(* Logix 5000 project; controller Modbus_TCP_Client_Example vendor 1 type 14 code 154 rev 32.15; software revision 32.05; part 5 of 10 *)

ADD_ON_INSTRUCTION AMP_Normal_Stop   (* revision 1.0 *)
// Applied Motion - Stop/Kill using Normal Deceleration - AOI
// Help:
// The Normal Stop AOI is used to stop and kill the drive using the normal deceleration set by the DE command.
VAR_IN_OUT
   Input : DINT[14]; {required}   // Drive Input Assembly
   Output : DINT[16]; {required}   // Drive Output Assembly
        [0]   // Command Word
        [10]   // Data/Register 1
        [11]   // Data/Register 2
        [1]   // Jog Speed (0.25 rev/min)
        [2]   // Jog Acceleration (10 rev/s/s)
        [3]   // Jog Deceleration (10 rev/s/s)
        [4]   // Point-to-Point Velocity (0.25 rev/min)
        [5]   // Point-to-Point Acceleration (10 rev/s/s)
        [6]   // Point-to-Point Deceleration (10 rev/s/s)
        [7]   // Point-to-Point Distance (Motor steps)
        [9]   // (2x ASCII Letters in 16 lower word)
END_VAR
VAR_INPUT
   RPI : DINT := 100; {visible}   // Drive Connection Request Packet Interval (milliseconds)
   Stop : BOOL; {required}   // Stop the drive axis
END_VAR
VAR_OUTPUT
   Sent : BOOL; {access Read Only, visible}   // Stop has been sent to drive
   In_Progress : BOOL; {access Read Only, visible}   // Stop in progress
   Done : BOOL; {access Read Only, visible}   // Stop completed without errors - Servo is not moving
   Error : BOOL; {access Read Only, visible}   // Stop failed - drive not ready or faulted
   State : DINT := 10; {access None}   // Internal state of progress
END_VAR
VAR
   Loc_StatusCode : AMP_Status_Word;
   Loc_CommandOff_Timer : TIMER;   // Timer to make sure command value was 0 before sending a new command
   Loc_CommandOn_Timer : TIMER;   // Timer to make sure command value is set long enough to be sent to servo
   Loc_Input_Assembly : AMP_Input_Assembly_v2; {access None}
   Loc_Stop_ONS : BOOL; {access None}
END_VAR

ROUTINE Logic   (* ladder *)
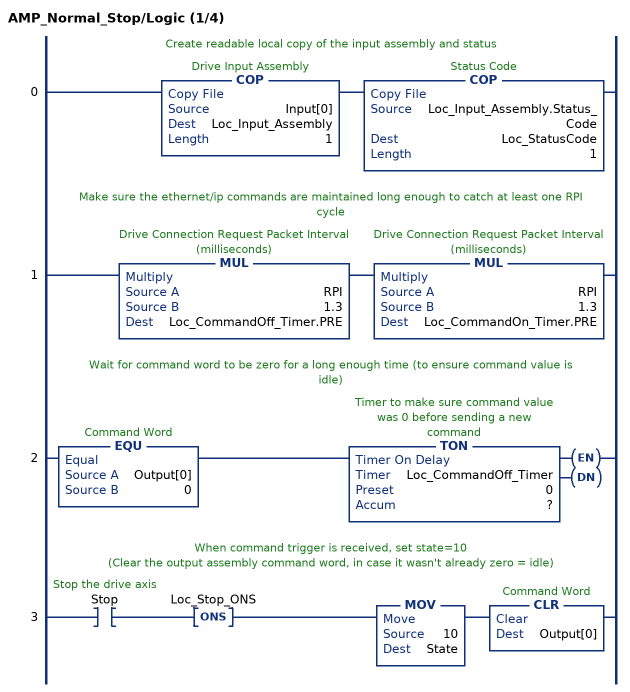
   // Create readable local copy of the input assembly and status
   0: COP(Input[0],Loc_Input_Assembly,1)COP(Loc_Input_Assembly.Status_Code,Loc_StatusCode,1);
   // Make sure the ethernet/ip commands are maintained long enough to catch at least one RPI cycle
   1: MUL(RPI,1.3,Loc_CommandOff_Timer.PRE)MUL(RPI,1.3,Loc_CommandOn_Timer.PRE);
   // Wait for command word to be zero for a long enough time (to ensure command value is idle)
   2: EQU(Output[0],0)TON(Loc_CommandOff_Timer,?,?);
   // When command trigger is received, set state=10
   // (Clear the output assembly command word, in case it wasn't already zero = idle)
   3: XIC(Stop)ONS(Loc_Stop_ONS)MOV(10,State)CLR(Output[0]);
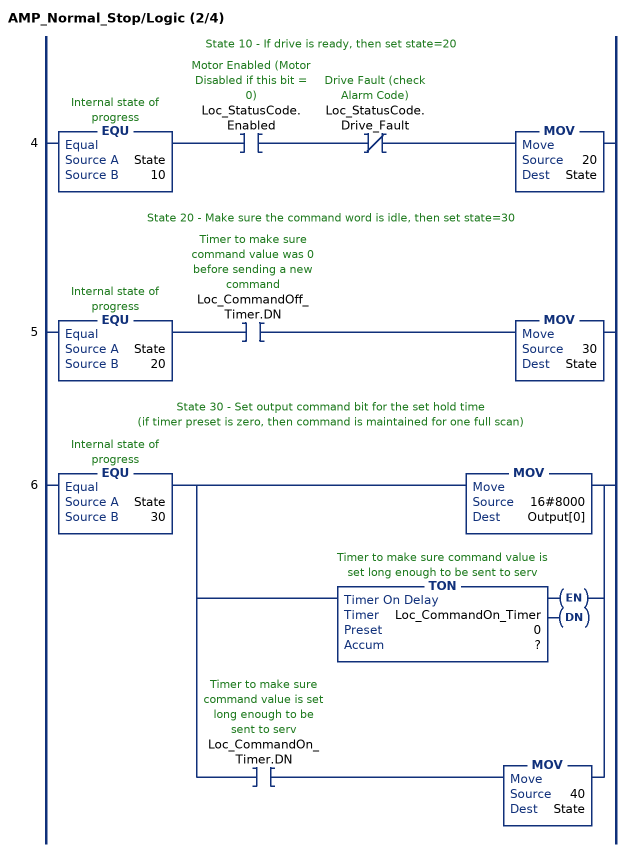
   // State 10 - If drive is ready, then set state=20
   4: EQU(State,10)XIC(Loc_StatusCode.Enabled)XIO(Loc_StatusCode.Drive_Fault)MOV(20,State);
   // State 20 - Make sure the command word is idle, then set state=30
   5: EQU(State,20)XIC(Loc_CommandOff_Timer.DN)MOV(30,State);
   // State 30 - Set output command bit for the set hold time
   // (if timer preset is zero, then command is maintained for one full scan)
   6: EQU(State,30)[MOV(16#8000,Output[0]) ,TON(Loc_CommandOn_Timer,?,?) ,XIC(Loc_CommandOn_Timer.DN) MOV(40,State) ];
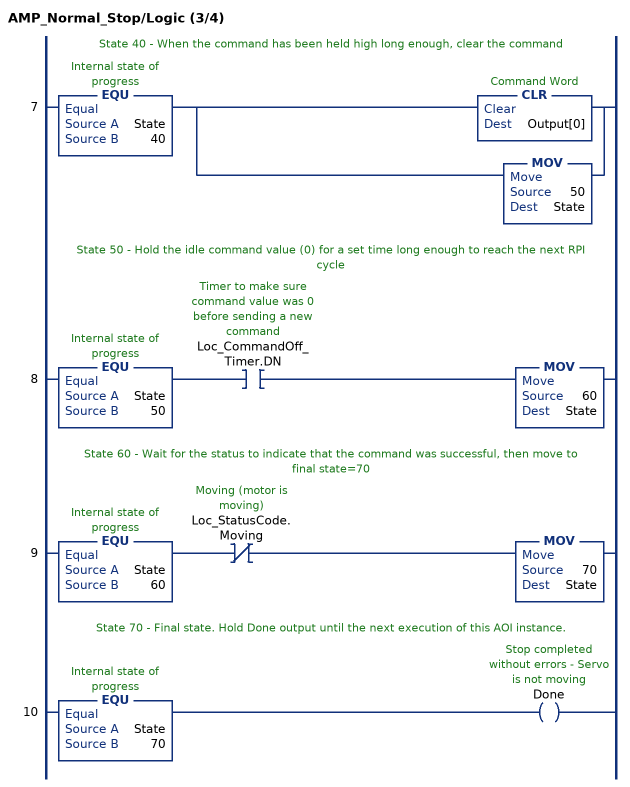
   // State 40 - When the command has been held high long enough, clear the command
   7: EQU(State,40)[CLR(Output[0]) ,MOV(50,State) ];
   // State 50 - Hold the idle command value (0) for a set time long enough to reach the next RPI cycle
   8: EQU(State,50)XIC(Loc_CommandOff_Timer.DN)MOV(60,State);
   // State 60 - Wait for the status to indicate that the command was successful, then move to final state=70
   9: EQU(State,60)XIO(Loc_StatusCode.Moving)MOV(70,State);
   // State 70 - Final state. Hold Done output until the next execution of this AOI instance.
   10: EQU(State,70)OTE(Done);
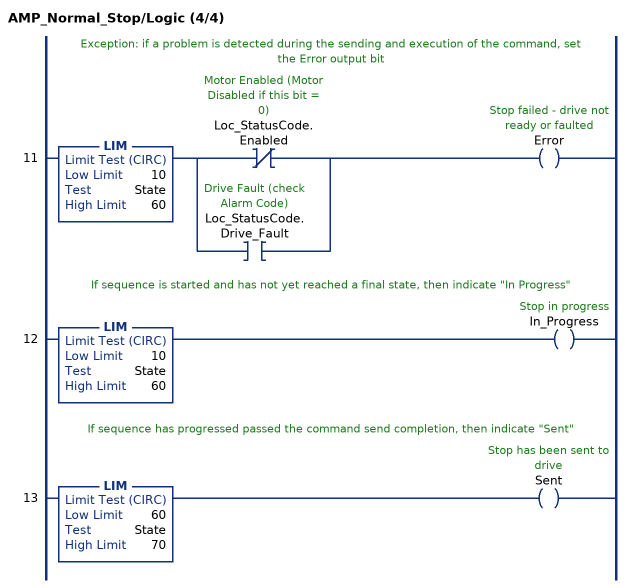
   // Exception: if a problem is detected during the sending and execution of the command, set the Error output bit
   11: LIM(10,State,60)[XIO(Loc_StatusCode.Enabled) ,XIC(Loc_StatusCode.Drive_Fault) ]OTE(Error);
   // If sequence is started and has not yet reached a final state, then indicate "In Progress"
   12: LIM(10,State,60)OTE(In_Progress);
   // If sequence has progressed passed the command send completion, then indicate "Sent"
   13: LIM(60,State,70)OTE(Sent);
END_ROUTINE
END_ADD_ON_INSTRUCTION

ADD_ON_INSTRUCTION AMP_Normal_Stop_Servo   (* revision 1.0, vendor Applied Motion Products Inc. *)
// Applied Motion - Stop/Kill using Normal Deceleration - AOI
// Help:
// This AOI Stops the Motor Jogging/Moving using Deceleration(SKD).
VAR_IN_OUT
   Input : DINT[20]; {required}   // Drive Input Assembly
        [16]   // Analog_Input1
        [4]   // Alarm_Code
        [0]   // Control_Word_Received
        [10]   // Position_Error
        [11]   // Actual_Velocity_RPS
        [12]   // Digital_Outputs
        [13]   // Digital_Inputs
        [14]   // Analog_Output1
        [15]   // Analog_Output2
        [17]   // Analog_Input2
        [18]   // Torque_Limit
        [19]   // Second_Encoder_Speed
        [1]   // OpCode1_Received
        [2]   // Control_Mode
        [3]   // Status_Code
        [5]   // Supply_Voltage
        [6]   // Applied_Torque
        [7]   // Drive_Temperature
        [8]   // Encoder_Position
        [9]   // Second_Encoder_Position
   Output : DINT[11]; {required}   // Drive Output Assembly
        [10]   // Reserved
        [4]   // Target Velocity
        [0]   // Control Word
        [3]   // Target Pos
        [1]   // OpCode 1
        [2]   // OpCode 2
        [5]   // Porifle Acceleration
        [6]   // Profile Deceleration
        [7]   // Target Torque
        [8]   // OpCode 3
        [9]   // OpCode 4
END_VAR
VAR_INPUT
   Stop : BOOL; {required}   // Stop the drive axis (on rising edge)
END_VAR
VAR_OUTPUT
   Sent : BOOL; {access Read Only, visible}   // Stop has been sent to drive
   In_Progress : BOOL; {access Read Only, visible}   // Stop in progress
   Done : BOOL; {access Read Only, visible}   // Stop completed without errors - Servo is not moving
   Error : BOOL; {access Read Only, visible}   // Stop failed - drive not ready or faulted
   State : DINT := 10; {access Read Only}   // Internal state of progress
END_VAR
VAR
   Loc_Stop_ONS : BOOL;
   Loc_StatusCode : AMP_Status_Word_Servo; {access None}
   Loc_Input_Assembly : AMP_Input_Assembly_Servo_v2; {access None}
END_VAR

ROUTINE Logic   (* ladder *)
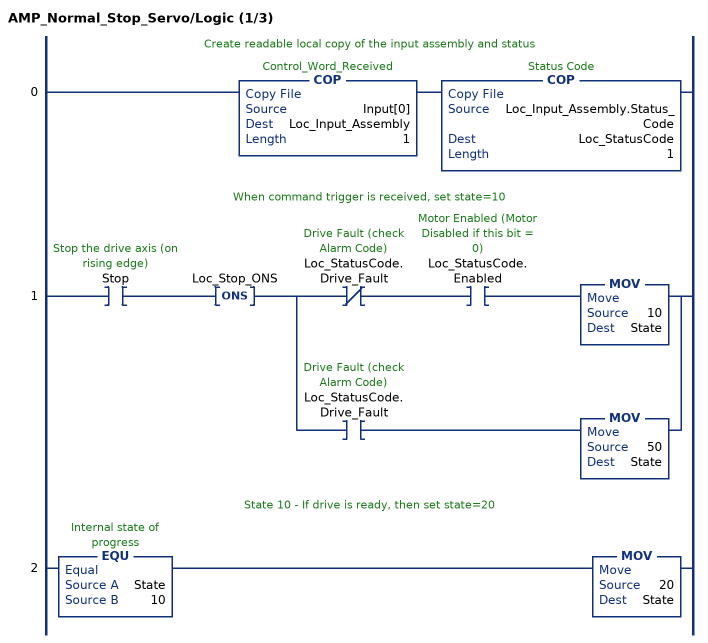
   // Create readable local copy of the input assembly and status
   0: COP(Input[0],Loc_Input_Assembly,1)COP(Loc_Input_Assembly.Status_Code,Loc_StatusCode,1);
   // When command trigger is received, set state=10
   1: XIC(Stop)ONS(Loc_Stop_ONS)[XIO(Loc_StatusCode.Drive_Fault) XIC(Loc_StatusCode.Enabled) MOV(10,State) ,XIC(Loc_StatusCode.Drive_Fault) MOV(50,State) ];
   // State 10 - If drive is ready, then set state=20
   2: EQU(State,10)MOV(20,State);
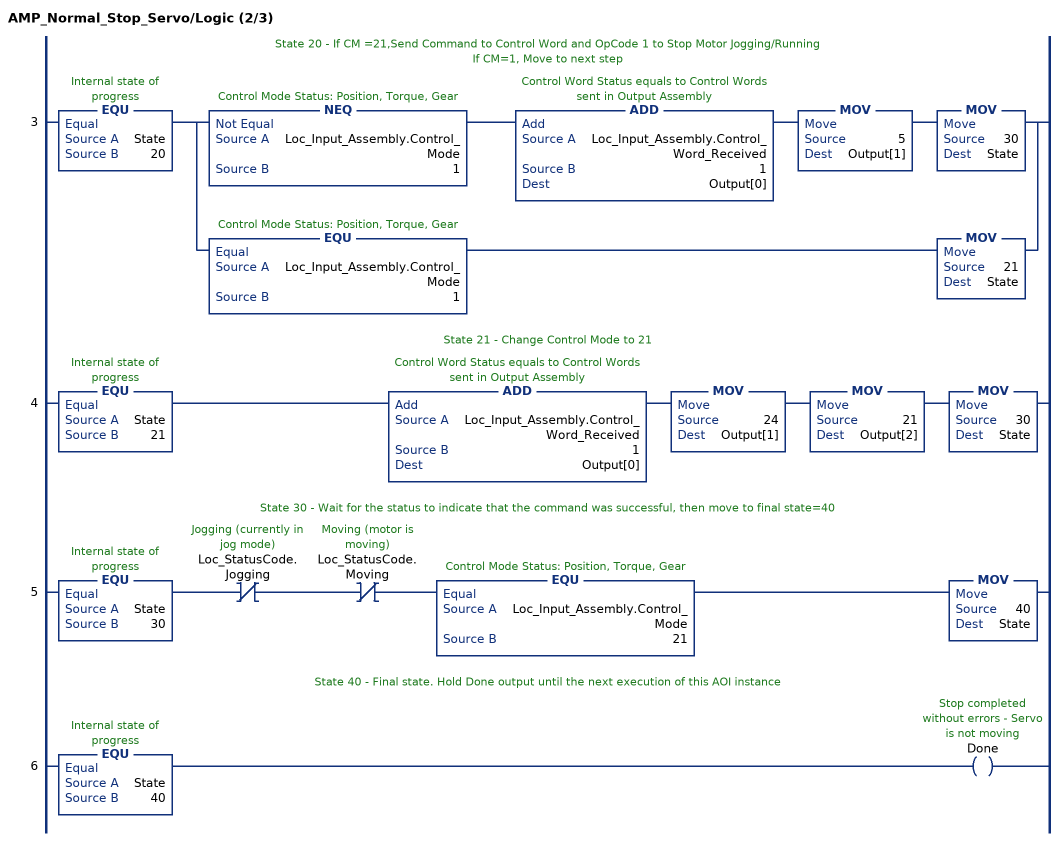
   // State 20 - If CM =21,Send Command to Control Word and OpCode 1 to Stop Motor Jogging/Running
   // If CM=1, Move to next step
   3: EQU(State,20)[NEQ(Loc_Input_Assembly.Control_Mode,1) ADD(Loc_Input_Assembly.Control_Word_Received,1,Output[0]) MOV(5,Output[1]) MOV(30,State) ,EQU(Loc_Input_Assembly.Control_Mode,1) MOV(21,State) ];
   // State 21 - Change Control Mode to 21
   4: EQU(State,21)ADD(Loc_Input_Assembly.Control_Word_Received,1,Output[0])MOV(24,Output[1])MOV(21,Output[2])MOV(30,State);
   // State 30 - Wait for the status to indicate that the command was successful, then move to final state=40
   5: EQU(State,30)XIO(Loc_StatusCode.Jogging)XIO(Loc_StatusCode.Moving)EQU(Loc_Input_Assembly.Control_Mode,21)MOV(40,State);
   // State 40 - Final state. Hold Done output until the next execution of this AOI instance
   6: EQU(State,40)OTE(Done);
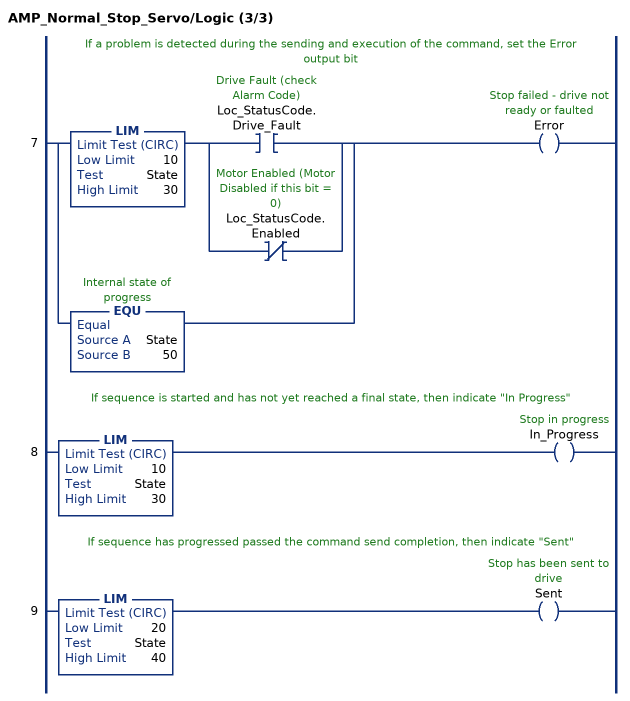
   // If a problem is detected during the sending and execution of the command, set the Error output bit
   7: [LIM(10,State,30) [XIC(Loc_StatusCode.Drive_Fault) ,XIO(Loc_StatusCode.Enabled) ] ,EQU(State,50) ]OTE(Error);
   // If sequence is started and has not yet reached a final state, then indicate "In Progress"
   8: LIM(10,State,30)OTE(In_Progress);
   // If sequence has progressed passed the command send completion, then indicate "Sent"
   9: LIM(20,State,40)OTE(Sent);
END_ROUTINE
END_ADD_ON_INSTRUCTION

ADD_ON_INSTRUCTION AMP_Point_to_Point_FC_Servo   (* revision 1.0, vendor Applied Motion Products Inc. *)
// Applied Motion - Point to Point Move with Speed Change AOI
// Help:
// The Point-to-Point Move with Speed Change AOI executes a feed to length (relative move) with a speed change after an initial travel distance (FC command).
VAR_IN_OUT
   Input : DINT[20]; {required}   // Drive Input Assembly
        [16]   // Analog_Input1
        [4]   // Alarm_Code
        [0]   // Control_Word_Received
        [10]   // Position_Error
        [11]   // Actual_Velocity_RPS
        [12]   // Digital_Outputs
        [13]   // Digital_Inputs
        [14]   // Analog_Output1
        [15]   // Analog_Output2
        [17]   // Analog_Input2
        [18]   // Torque_Limit
        [19]   // Second_Encoder_Speed
        [1]   // OpCode1_Received
        [2]   // Control_Mode
        [3]   // Status_Code
        [5]   // Supply_Voltage
        [6]   // Applied_Torque
        [7]   // Drive_Temperature
        [8]   // Encoder_Position
        [9]   // Second_Encoder_Position
   Output : DINT[11]; {required}   // Drive Output Assembly
        [10]   // Reserved
        [4]   // Target Velocity
        [0]   // Control Word
        [3]   // Target Pos
        [1]   // OpCode 1
        [2]   // OpCode 2
        [5]   // Porifle Acceleration
        [6]   // Profile Deceleration
        [7]   // Target Torque
        [8]   // OpCode 3
        [9]   // OpCode 4
END_VAR
VAR_INPUT
   Start : BOOL; {required}   // Start the Move
   Distance : DINT; {required}   // Distance to Move (steps, negative = reverse)
   Speed : REAL; {required}   // Velocity of Move (rev/sec)
   Acc : REAL; {required}   // Acceleration of Move (rev/s/s)
   Dec : REAL; {required}   // Deceleration (rev/s/s)
   Change_Distance : DINT; {required}   // Change Distance (steps)
   Change_Speed : REAL; {required}   // Velocity Change (rev/s)
END_VAR
VAR_OUTPUT
   Sent : BOOL; {access Read Only, visible}   // Move has been sent to drive
   In_Progress : BOOL; {access Read Only, visible}   // Move in progress
   Done : BOOL; {access Read Only, visible}   // Move completed without errors - desired position reached
   Error : BOOL; {access Read Only, visible}   // Move failed to complete - drive not ready or faulted
   State : DINT := 10; {access Read Only}   // Internal state of progress
END_VAR
VAR
   Loc_Command_Timeout : TIMER := (PRE := 2000); {access None}   // Timer to output fault if command is not Done
   Loc_StatusCode : AMP_Status_Word_Servo; {access None}
   Loc_Start_ONS : BOOL; {access None}
   Loc_Input_Assembly : AMP_Input_Assembly_Servo_v2; {access None}
   Loc_ChangeSpeed_Required : BOOL; {access None}
   Loc_ChangeDistance_Required : BOOL; {access None}
END_VAR

ROUTINE Logic   (* ladder *)
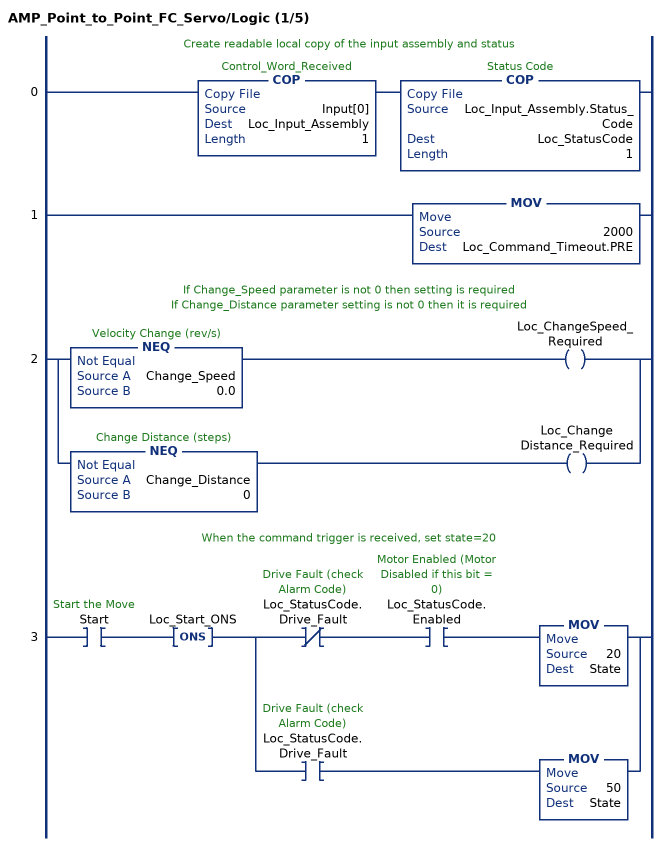
   // Create readable local copy of the input assembly and status
   0: COP(Input[0],Loc_Input_Assembly,1)COP(Loc_Input_Assembly.Status_Code,Loc_StatusCode,1);
   1: MOV(2000,Loc_Command_Timeout.PRE);
   // If Change_Speed parameter is not 0 then setting is required
   // If Change_Distance parameter setting is not 0 then it is required
   2: [NEQ(Change_Speed,0.0) OTE(Loc_ChangeSpeed_Required) ,NEQ(Change_Distance,0) OTE(Loc_ChangeDistance_Required) ];
   // When the command trigger is received, set state=20
   3: XIC(Start)ONS(Loc_Start_ONS)[XIO(Loc_StatusCode.Drive_Fault) XIC(Loc_StatusCode.Enabled) MOV(20,State) ,XIC(Loc_StatusCode.Drive_Fault) MOV(50,State) ];
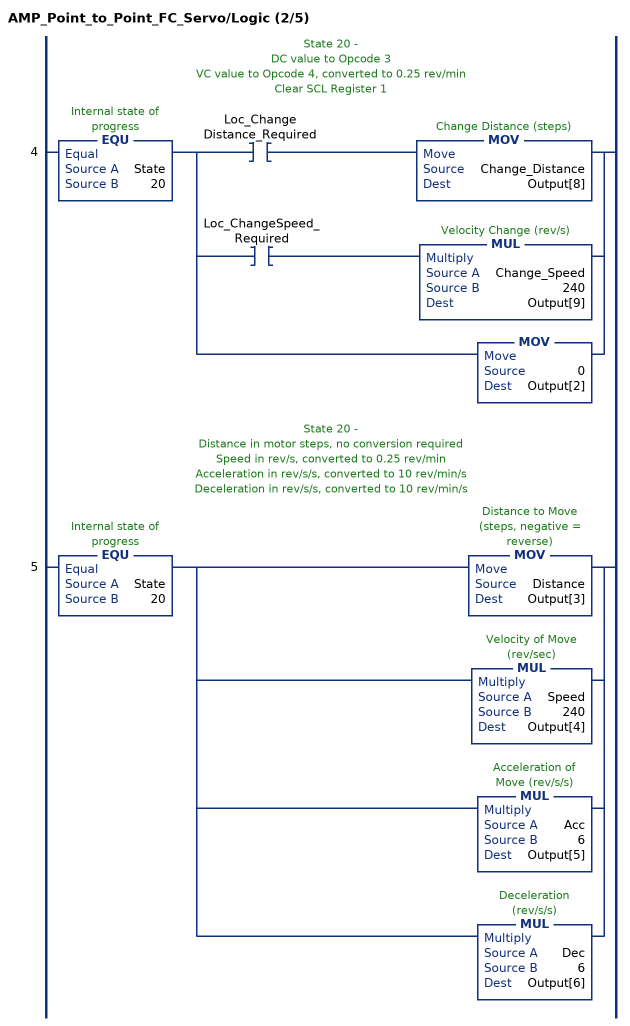
   // State 20 -
   // DC value to Opcode 3
   // VC value to Opcode 4, converted to 0.25 rev/min
   // Clear SCL Register 1
   4: EQU(State,20)[XIC(Loc_ChangeDistance_Required) MOV(Change_Distance,Output[8]) ,XIC(Loc_ChangeSpeed_Required) MUL(Change_Speed,240,Output[9]) ,MOV(0,Output[2]) ];
   // State 20 -
   // Distance in motor steps, no conversion required
   // Speed in rev/s, converted to 0.25 rev/min
   // Acceleration in rev/s/s, converted to 10 rev/min/s
   // Deceleration in rev/s/s, converted to 10 rev/min/s
   5: EQU(State,20)[MOV(Distance,Output[3]) ,MUL(Speed,240,Output[4]) ,MUL(Acc,6,Output[5]) ,MUL(Dec,6,Output[6]) ];
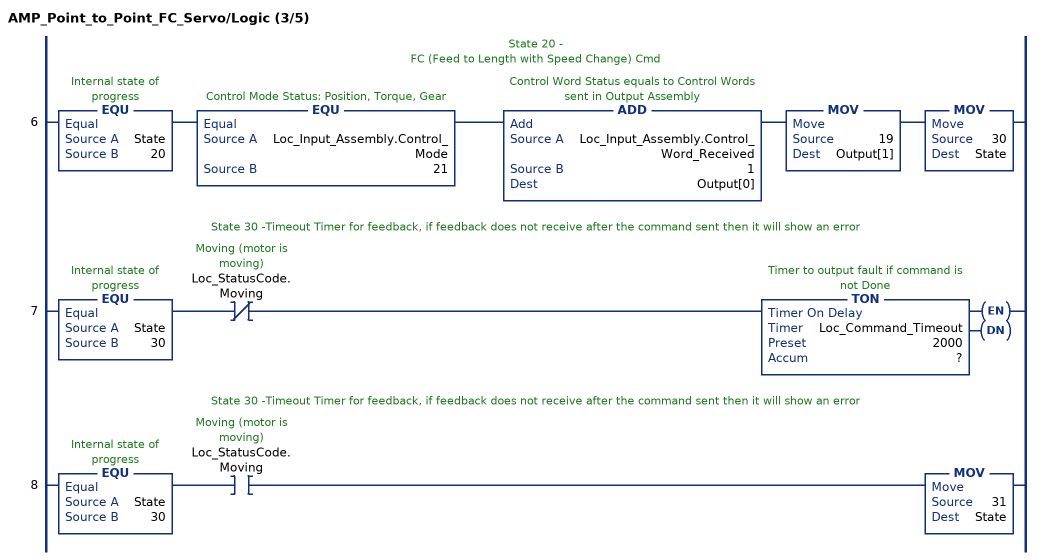
   // State 20 -
   // FC (Feed to Length with Speed Change) Cmd
   6: EQU(State,20)EQU(Loc_Input_Assembly.Control_Mode,21)ADD(Loc_Input_Assembly.Control_Word_Received,1,Output[0])MOV(19,Output[1])MOV(30,State);
   // State 30 -Timeout Timer for feedback, if feedback does not receive after the command sent then it will show an error
   7: EQU(State,30)XIO(Loc_StatusCode.Moving)TON(Loc_Command_Timeout,?,?);
   // State 30 -Timeout Timer for feedback, if feedback does not receive after the command sent then it will show an error
   8: EQU(State,30)XIC(Loc_StatusCode.Moving)MOV(31,State);
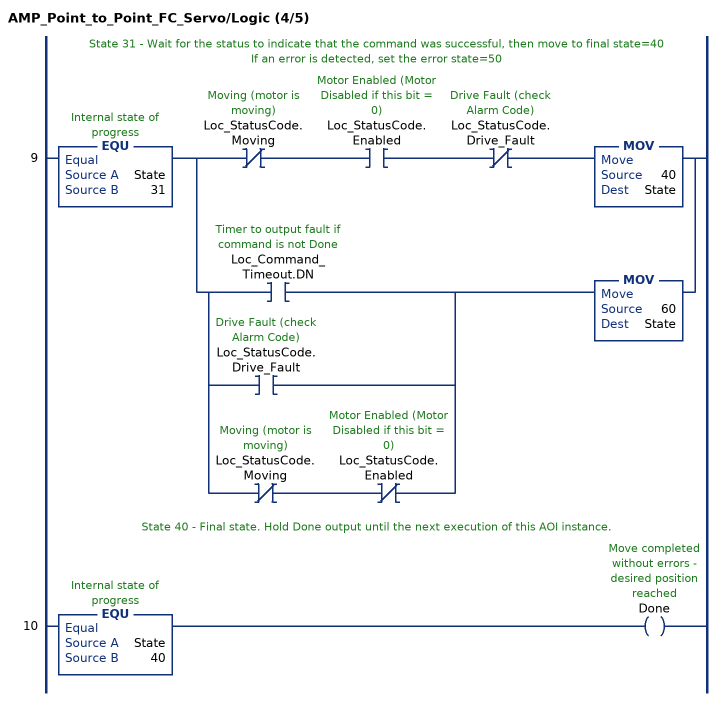
   // State 31 - Wait for the status to indicate that the command was successful, then move to final state=40
   // If an error is detected, set the error state=50
   9: EQU(State,31)[XIO(Loc_StatusCode.Moving) XIC(Loc_StatusCode.Enabled) XIO(Loc_StatusCode.Drive_Fault) MOV(40,State) ,[XIC(Loc_Command_Timeout.DN) ,XIC(Loc_StatusCode.Drive_Fault) ,XIO(Loc_StatusCode.Moving) XIO(Loc_StatusCode.Enabled) ] MOV(60,State) ];
   // State 40 - Final state. Hold Done output until the next execution of this AOI instance.
   10: EQU(State,40)OTE(Done);
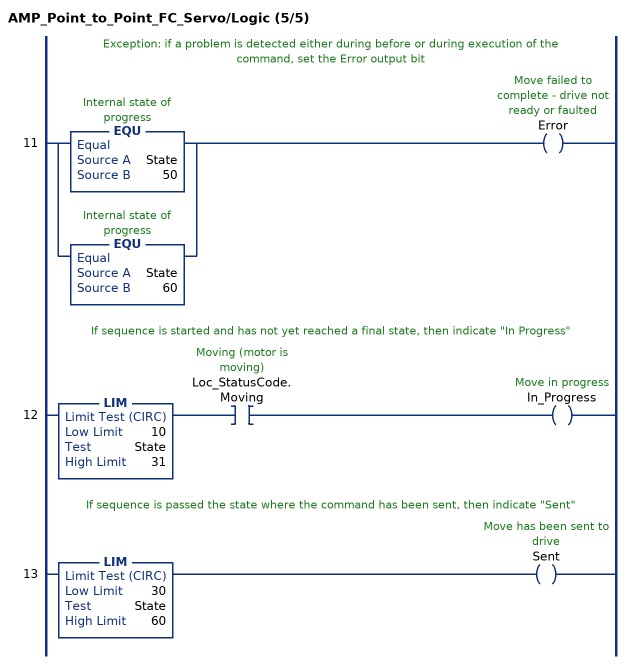
   // Exception: if a problem is detected either during before or during execution of the command, set the Error output bit
   11: [EQU(State,50) ,EQU(State,60) ]OTE(Error);
   // If sequence is started and has not yet reached a final state, then indicate "In Progress"
   12: LIM(10,State,31)XIC(Loc_StatusCode.Moving)OTE(In_Progress);
   // If sequence is passed the state where the command has been sent, then indicate "Sent"
   13: LIM(30,State,60)OTE(Sent);
END_ROUTINE
END_ADD_ON_INSTRUCTION

ADD_ON_INSTRUCTION AMP_Point_to_Point_IO   (* revision 1.0 *)
// Applied Motion - Point to Point Move with IO AOI
// Help:
// The Point-to-Point Move with I/O AOI executes moves involving up to 2 Input conditions and a possible output state change. The move variant can be any of the following:
// - FS - Feed to Sensor
// - FD - Feed to Double Sensor
// - FM - Feed to Sensor with Mask Distance
// - FY - Feed to Sensor with Safety Distance
// - FO - Feed to Length and Set Output
// - FE - Follow Encoder
// - SH - Seek Home
// All seven (7) of the above variants need exactly one I/O point except for FD which requires a second I/O point to be specified in the parameters.
VAR_IN_OUT
   Input : DINT[14]; {required}   // Drive Input Assembly
   Output : DINT[16]; {required}   // Drive Output Assembly
        [0]   // Command Word
        [10]   // Data/Register 1
        [11]   // Data/Register 2
        [1]   // Jog Speed (0.25 rev/min)
        [2]   // Jog Acceleration (10 rev/s/s)
        [3]   // Jog Deceleration (10 rev/s/s)
        [4]   // Point-to-Point Velocity (0.25 rev/min)
        [5]   // Point-to-Point Acceleration (10 rev/s/s)
        [6]   // Point-to-Point Deceleration (10 rev/s/s)
        [7]   // Point-to-Point Distance (Motor steps)
        [9]   // (2x ASCII Letters in 16 lower word)
END_VAR
VAR_INPUT
   RPI : DINT := 100; {visible}   // Drive Connection Request Packet Interval (milliseconds)
   Start : BOOL; {required}   // Start the Move
   Command : INT := 'FE'; {required}   // Command variant: FS/FD/FY/FM/FO/SH/FE
   IO1_Number : DINT; {required}   // Main Input/Output Number (0 = Encoder index, 1-8 = In/Out 1-8)
   IO1_Condition : SINT := 'R'; {required}   // Main Input/Output Condition/State H/L/R/F (High/Low/Rising Edge/Falling Edge)
   IO2_Number : DINT; {required}   // Second Input/Output Number (0 = Encoder index, 1-8 = In/Out 1-8)
   IO2_Condition : SINT; {required}   // Second Input/Output Condition/State H/L/R/F (High/Low/Rising Edge/Falling Edge)
   IO_Connector : DINT := 1; {required}   // I/O Connector (1=IN/OUT 1, 2=IN/OUT 2)
   Distance : DINT; {required}   // Distance to Move (negative = reverse)
   Speed : REAL; {required}   // Velocity of Move (rev/min)
   Acc : REAL; {required}   // Acceleration of Move (rev/s/s)
   Dec : REAL; {required}   // Deceleration (rev/s/s)
   Change_Distance : DINT; {required}   // Change Distance (steps, FY/FM/FO only)
   Change_Speed : REAL; {required}   // Velocity Change (rev/s) (FD only)
END_VAR
VAR_OUTPUT
   Sent : BOOL; {access Read Only, visible}   // Move has been sent to drive
   In_Progress : BOOL; {access Read Only, visible}   // Move in progress
   Done : BOOL; {access Read Only, visible}   // Move completed without errors - desired position reached
   Error : BOOL; {access Read Only, visible}   // Move failed to complete - drive not ready or faulted
   State : DINT := 10; {access Read Only}   // Internal state of progress
END_VAR
VAR
   Loc_StatusCode : AMP_Status_Word;
   Loc_CommandOff_Timer : TIMER;   // Timer to make sure command value was 0 before sending a new command
   Loc_CommandOn_Timer : TIMER;   // Timer to make sure command value is set long enough to be sent to drive
   Loc_Input_Assembly : AMP_Input_Assembly_v2; {access None}
   Loc_Start_ONS : BOOL; {access None}
   Loc_ChangeSpeed_Required : BOOL; {access None}
   Loc_ChangeDistance_Required : BOOL; {access None}
   Loc_IO1_Condition_Encoded : INT; {access None}
   Loc_IO1_Number_Encoded : INT; {access None}
   Loc_IO2_Condition_Encoded : INT; {access None}
   Loc_IO2_Number_Encoded : INT; {access None}
END_VAR

ROUTINE Logic   (* ladder *)
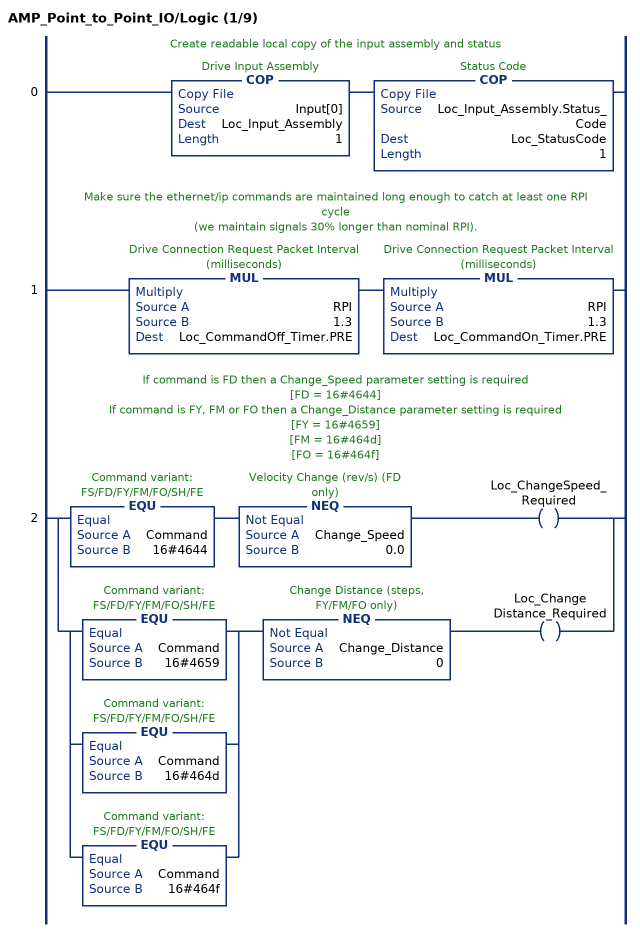
   // Create readable local copy of the input assembly and status
   0: COP(Input[0],Loc_Input_Assembly,1)COP(Loc_Input_Assembly.Status_Code,Loc_StatusCode,1);
   // Make sure the ethernet/ip commands are maintained long enough to catch at least one RPI cycle
   // (we maintain signals 30% longer than nominal RPI).
   1: MUL(RPI,1.3,Loc_CommandOff_Timer.PRE)MUL(RPI,1.3,Loc_CommandOn_Timer.PRE);
   // If command is FD then a Change_Speed parameter setting is required
   // [FD = 16#4644]
   // If command is FY, FM or FO then a Change_Distance parameter setting is required
   // [FY = 16#4659]
   // [FM = 16#464d]
   // [FO = 16#464f]
   2: [EQU(Command,16#4644) NEQ(Change_Speed,0.0) OTE(Loc_ChangeSpeed_Required) ,[EQU(Command,16#4659) ,EQU(Command,16#464d) ,EQU(Command,16#464f) ] NEQ(Change_Distance,0) OTE(Loc_ChangeDistance_Required) ];
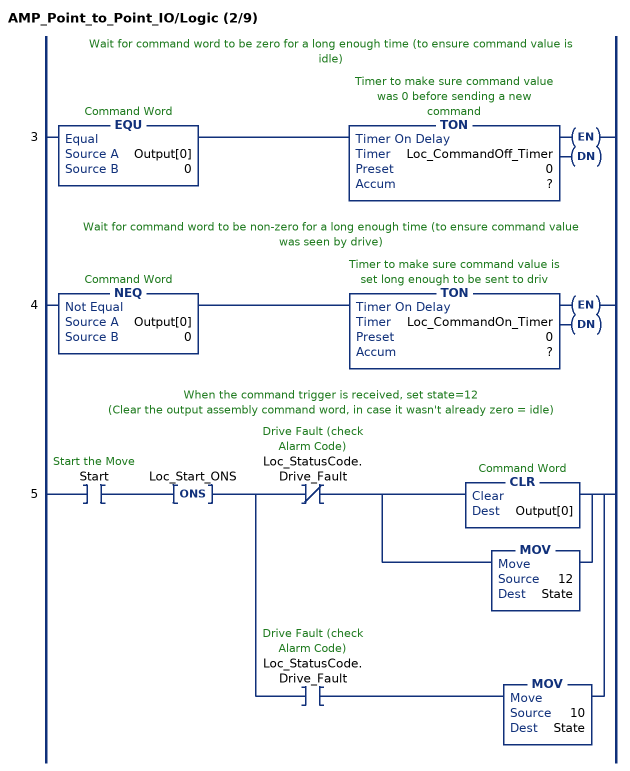
   // Wait for command word to be zero for a long enough time (to ensure command value is idle)
   3: EQU(Output[0],0)TON(Loc_CommandOff_Timer,?,?);
   // Wait for command word to be non-zero for a long enough time (to ensure command value was seen by drive)
   4: NEQ(Output[0],0)TON(Loc_CommandOn_Timer,?,?);
   // When the command trigger is received, set state=12
   // (Clear the output assembly command word, in case it wasn't already zero = idle)
   5: XIC(Start)ONS(Loc_Start_ONS)[XIO(Loc_StatusCode.Drive_Fault) [CLR(Output[0]) ,MOV(12,State) ] ,XIC(Loc_StatusCode.Drive_Fault) MOV(10,State) ];
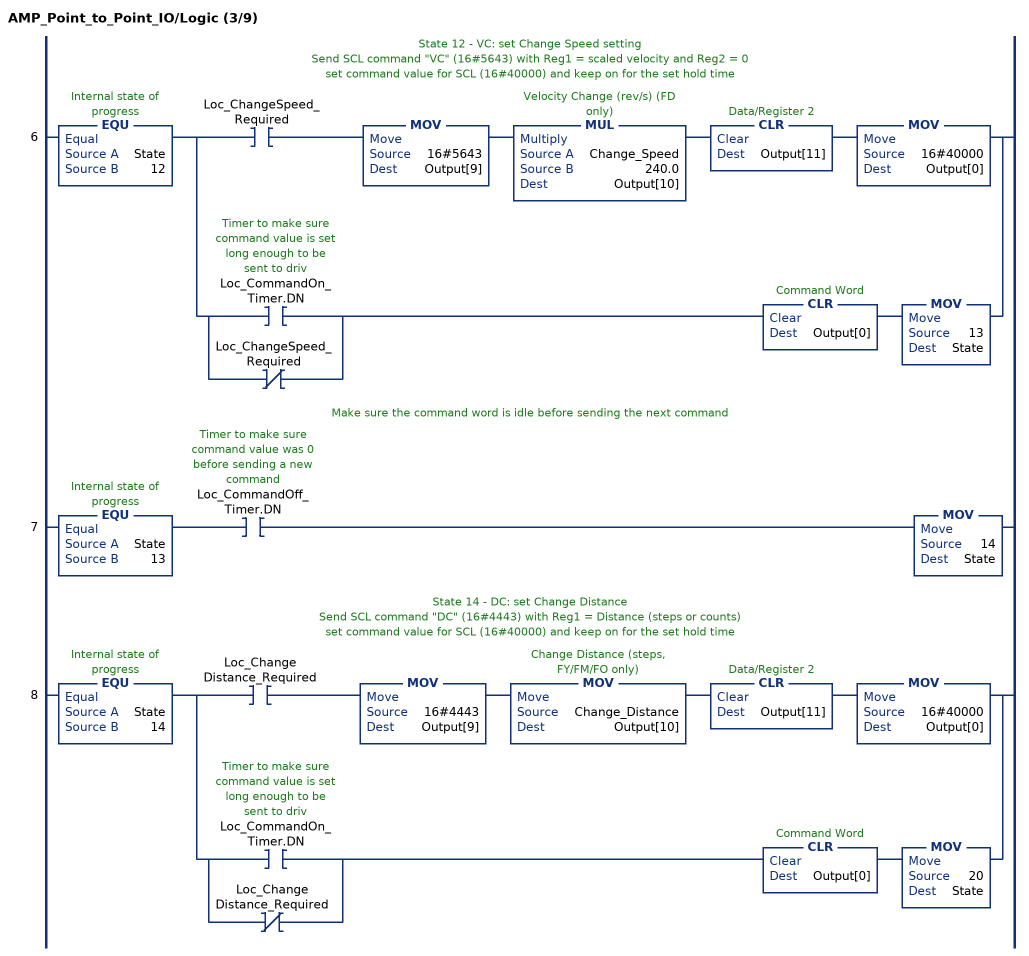
   // State 12 - VC: set Change Speed setting
   // Send SCL command "VC" (16#5643) with Reg1 = scaled velocity and Reg2 = 0
   // set command value for SCL (16#40000) and keep on for the set hold time
   6: EQU(State,12)[XIC(Loc_ChangeSpeed_Required) MOV(16#5643,Output[9]) MUL(Change_Speed,240.0,Output[10]) CLR(Output[11]) MOV(16#40000,Output[0]) ,[XIC(Loc_CommandOn_Timer.DN) ,XIO(Loc_ChangeSpeed_Required) ] CLR(Output[0]) MOV(13,State) ];
   // Make sure the command word is idle before sending the next command
   7: EQU(State,13)XIC(Loc_CommandOff_Timer.DN)MOV(14,State);
   // State 14 - DC: set Change Distance
   // Send SCL command "DC" (16#4443) with Reg1 = Distance (steps or counts)
   // set command value for SCL (16#40000) and keep on for the set hold time
   8: EQU(State,14)[XIC(Loc_ChangeDistance_Required) MOV(16#4443,Output[9]) MOV(Change_Distance,Output[10]) CLR(Output[11]) MOV(16#40000,Output[0]) ,[XIC(Loc_CommandOn_Timer.DN) ,XIO(Loc_ChangeDistance_Required) ] CLR(Output[0]) MOV(20,State) ];
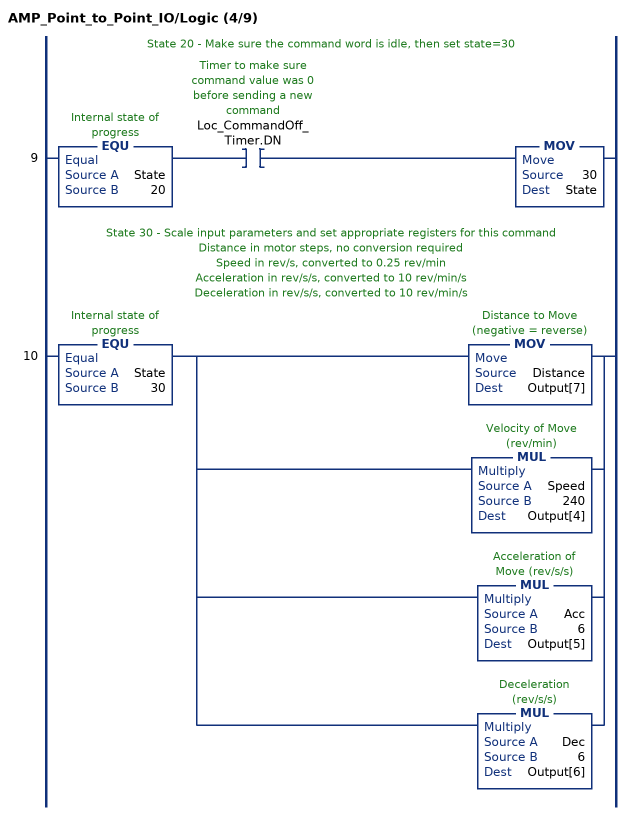
   // State 20 - Make sure the command word is idle, then set state=30
   9: EQU(State,20)XIC(Loc_CommandOff_Timer.DN)MOV(30,State);
   // State 30 - Scale input parameters and set appropriate registers for this command
   // Distance in motor steps, no conversion required
   // Speed in rev/s, converted to 0.25 rev/min
   // Acceleration in rev/s/s, converted to 10 rev/min/s
   // Deceleration in rev/s/s, converted to 10 rev/min/s
   10: EQU(State,30)[MOV(Distance,Output[7]) ,MUL(Speed,240,Output[4]) ,MUL(Acc,6,Output[5]) ,MUL(Dec,6,Output[6]) ];
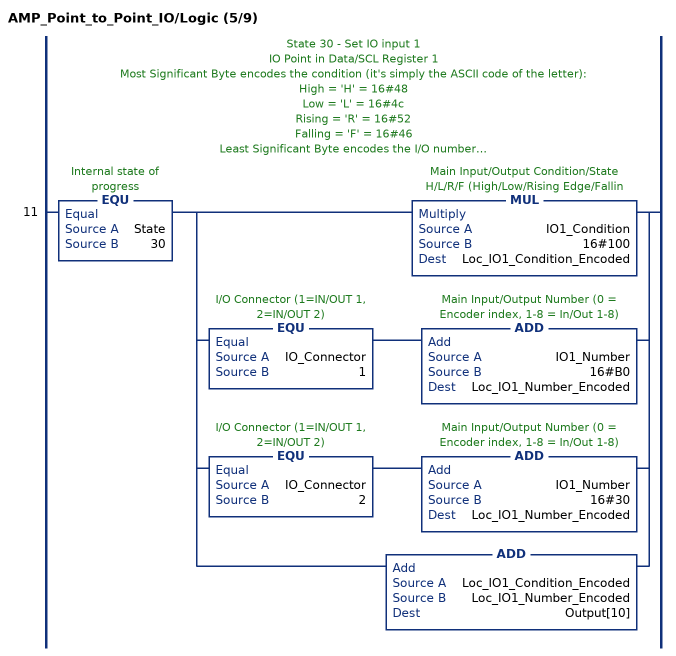
   // State 30 - Set IO input 1
   // IO Point in Data/SCL Register 1
   // Most Significant Byte encodes the condition (it's simply the ASCII code of the letter):
   // High = 'H' = 16#48
   // Low = 'L' = 16#4c
   // Rising = 'R' = 16#52
   // Falling = 'F' = 16#46
   // Least Significant Byte encodes the I/O number:
   // 0xB0-0xBC for connector 1 (IN/OUT1) depending on provided I/O number 0-12 (0=encoder)
   // 0x30-0x3C for connector 2 (IN/OUT2) depending on provided I/O numbers 0-12 (0=encoder)
   11: EQU(State,30)[MUL(IO1_Condition,16#100,Loc_IO1_Condition_Encoded) ,EQU(IO_Connector,1) ADD(IO1_Number,16#B0,Loc_IO1_Number_Encoded) ,EQU(IO_Connector,2) ADD(IO1_Number,16#30,Loc_IO1_Number_Encoded) ,ADD(Loc_IO1_Condition_Encoded,Loc_IO1_Number_Encoded,Output[10]) ];
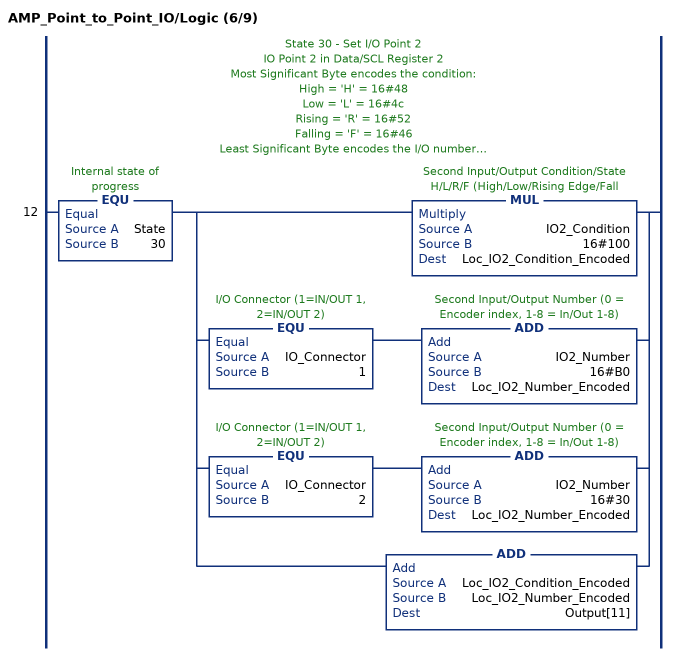
   // State 30 - Set I/O Point 2
   // IO Point 2 in Data/SCL Register 2
   // Most Significant Byte encodes the condition:
   // High = 'H' = 16#48
   // Low = 'L' = 16#4c
   // Rising = 'R' = 16#52
   // Falling = 'F' = 16#46
   // Least Significant Byte encodes the I/O number:
   // 0xB0-0xBC for connector 1 (IN/OUT1) depending on provided I/O number 0-12 (0=encoder)
   // 0x30-0x3C for connector 2 (IN/OUT2) depending on provided I/O numbers 0-12 (0=encoder)
   12: EQU(State,30)[MUL(IO2_Condition,16#100,Loc_IO2_Condition_Encoded) ,EQU(IO_Connector,1) ADD(IO2_Number,16#B0,Loc_IO2_Number_Encoded) ,EQU(IO_Connector,2) ADD(IO2_Number,16#30,Loc_IO2_Number_Encoded) ,ADD(Loc_IO2_Condition_Encoded,Loc_IO2_Number_Encoded,Output[11]) ];
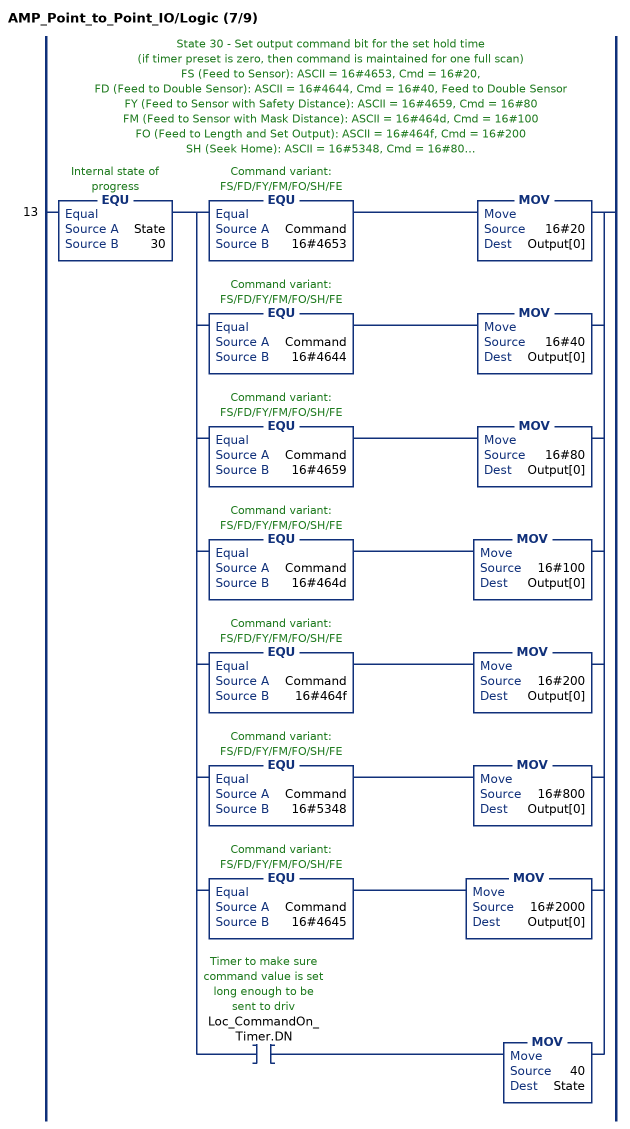
   // State 30 - Set output command bit for the set hold time
   // (if timer preset is zero, then command is maintained for one full scan)
   // FS (Feed to Sensor): ASCII = 16#4653, Cmd = 16#20,
   // FD (Feed to Double Sensor): ASCII = 16#4644, Cmd = 16#40, Feed to Double Sensor
   // FY (Feed to Sensor with Safety Distance): ASCII = 16#4659, Cmd = 16#80
   // FM (Feed to Sensor with Mask Distance): ASCII = 16#464d, Cmd = 16#100
   // FO (Feed to Length and Set Output): ASCII = 16#464f, Cmd = 16#200
   // SH (Seek Home): ASCII = 16#5348, Cmd = 16#800
   // FE (Follow Encoder): ASCII = 16#4645, Cmd = 16#2000
   13: EQU(State,30)[[EQU(Command,16#4653) MOV(16#20,Output[0]) ,EQU(Command,16#4644) MOV(16#40,Output[0]) ,EQU(Command,16#4659) MOV(16#80,Output[0]) ,EQU(Command,16#464d) MOV(16#100,Output[0]) ,EQU(Command,16#464f) MOV(16#200,Output[0]) ,EQU(Command,16#5348) MOV(16#800,Output[0]) ,EQU(Command,16#4645) MOV(16#2000,Output[0]) ] ,XIC(Loc_CommandOn_Timer.DN) MOV(40,State) ];
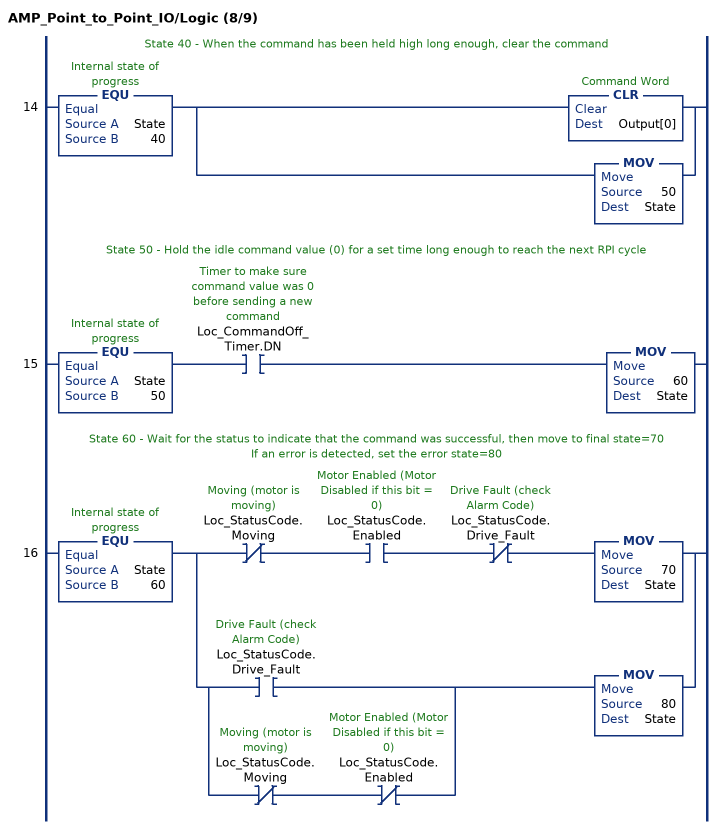
   // State 40 - When the command has been held high long enough, clear the command
   14: EQU(State,40)[CLR(Output[0]) ,MOV(50,State) ];
   // State 50 - Hold the idle command value (0) for a set time long enough to reach the next RPI cycle
   15: EQU(State,50)XIC(Loc_CommandOff_Timer.DN)MOV(60,State);
   // State 60 - Wait for the status to indicate that the command was successful, then move to final state=70
   // If an error is detected, set the error state=80
   16: EQU(State,60)[XIO(Loc_StatusCode.Moving) XIC(Loc_StatusCode.Enabled) XIO(Loc_StatusCode.Drive_Fault) MOV(70,State) ,[XIC(Loc_StatusCode.Drive_Fault) ,XIO(Loc_StatusCode.Moving) XIO(Loc_StatusCode.Enabled) ] MOV(80,State) ];
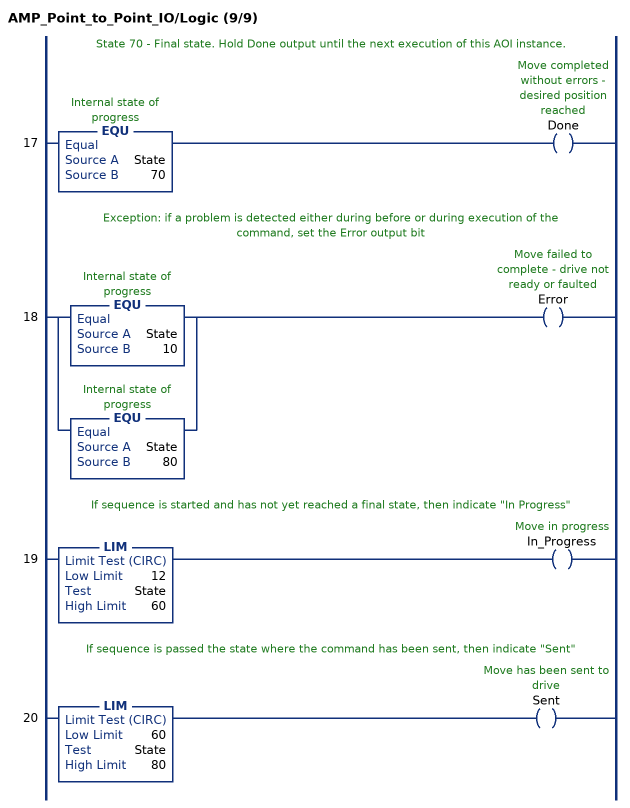
   // State 70 - Final state. Hold Done output until the next execution of this AOI instance.
   17: EQU(State,70)OTE(Done);
   // Exception: if a problem is detected either during before or during execution of the command, set the Error output bit
   18: [EQU(State,10) ,EQU(State,80) ]OTE(Error);
   // If sequence is started and has not yet reached a final state, then indicate "In Progress"
   19: LIM(12,State,60)OTE(In_Progress);
   // If sequence is passed the state where the command has been sent, then indicate "Sent"
   20: LIM(60,State,80)OTE(Sent);
END_ROUTINE
END_ADD_ON_INSTRUCTION
